# EPICS substitutions: iocBoot/iocAmptek/Amptek_SCAs.substitutions
file "$(MCA)/db/Amptek_SCAn.db"
{
pattern
{PORT,    P,           R,     M,    N}
{Amptek1, mcaTest:, Amptek1:, mca1, 0}
{Amptek1, mcaTest:, Amptek1:, mca1, 1}
{Amptek1, mcaTest:, Amptek1:, mca1, 2}
{Amptek1, mcaTest:, Amptek1:, mca1, 3}
{Amptek1, mcaTest:, Amptek1:, mca1, 4}
{Amptek1, mcaTest:, Amptek1:, mca1, 5}
{Amptek1, mcaTest:, Amptek1:, mca1, 6}
{Amptek1, mcaTest:, Amptek1:, mca1, 7}
}
